{attribute 'GeneratedUsingTerminal: EPP3744-0041-0016'}
{attribute addProperty BoxType "EPP3744-0041-0016"}
{attribute addProperty Id "EtcSlaveTerminalBaseDIG_InputsAT %I*DIG_Inputs_697E0EF26AI_Inputs_Channel_1AT %I*AI_Inputs_Channel_4521310411AI_Inputs_Channel_2AT %I*AI_Inputs_Channel_4521310411AI_Inputs_Channel_3AT %I*AI_Inputs_Channel_4521310411AI_Inputs_Channel_4AT %I*AI_Inputs_Channel_4521310411DEV_Inputs_DeviceAT %I*DEV_Inputs_Device_5F4E175E5DIG_OutputsAT %Q*DIG_Outputs_DE230DD52DEV_Outputs_DeviceAT %Q*DEV_Outputs_Device_59FFD2471WcStateAT %I*WcState_9091E0EB2InfoDataAT %I*InfoData_32EB74EA10"}
{attribute addProperty CRC "4099206104"}
{attribute addProperty Size "70"}
TYPE EPP3744_F454EBD8 EXTENDS EtcSlaveTerminalBase :
STRUCT
	{attribute addProperty Name "DIG_Inputs"}
	DIG_Inputs : DIG_Inputs_697E0EF2;
	{attribute addProperty Name "AI_Inputs_Channel_1"}
	AI_Inputs_Channel_1 : AI_Inputs_Channel_45213104;
	{attribute addProperty Name "AI_Inputs_Channel_2"}
	AI_Inputs_Channel_2 : AI_Inputs_Channel_45213104;
	{attribute addProperty Name "AI_Inputs_Channel_3"}
	AI_Inputs_Channel_3 : AI_Inputs_Channel_45213104;
	{attribute addProperty Name "AI_Inputs_Channel_4"}
	AI_Inputs_Channel_4 : AI_Inputs_Channel_45213104;
	{attribute addProperty Name "DEV_Inputs_Device"}
	DEV_Inputs_Device : DEV_Inputs_Device_5F4E175E;
	{attribute addProperty Name "DIG_Outputs"}
	DIG_Outputs : DIG_Outputs_DE230DD5;
	{attribute addProperty Name "DEV_Outputs_Device"}
	DEV_Outputs_Device : DEV_Outputs_Device_59FFD247;
	{attribute addProperty Name "WcState"}
	WcState : WcState_9091E0EB;
	{attribute addProperty Name "InfoData"}
	InfoData : InfoData_32EB74EA;
END_STRUCT
END_TYPE

(* stored: Version 1.2.0.0, ProductVersion 3.1.4024.9
   DUT EPP3744_F454EBD8: Id {dafb4fac-b82f-41ff-9758-a11a9f5d8a05} *)
